(* CODESYS project ST_MUX.project

Project tree, tasks and I/O mapping:
  Device : AC702, Shenzhen Inovance Technology Co., Ltd., version 3.5.11.51
    application Application
      libraries: Standard, * (System)
      task MainTask (cyclic, interval 4 ms, priority 2) calls PLC_PRG
      program PLC_PRG [ST]
      DifferentialMonitor
    HardWare Configuration
    Network Configuration
    Device Diagnosis
    Resources List
    ConfigStorage
    SoftMotion General Axis Pool
    LocalHSIO : 本地高速IO, 汇川技术股份有限公司, version 1.0.0.0
        unmapped channels: DigitalInput, DigitalOutput
    MODBUS_TCP : ModbusTCP本地从站, inovance, version 00.00.00.10
    HwConfiguratioinDevice : SystemConfig, Inovance, version 00.00.00.10
        settings: NetworkConfigArray.NetworkConfigArray.BusType = 10; NetworkConfigArray.NetworkConfigArray.RackSum = 1; NetworkConfigArray.NetworkConfigArray.HardwareConfigArray.HardwareConfigArray.RackNo = 1
*)

// Device/Application/PLC_PRG
PROGRAM PLC_PRG
VAR
	A1: BOOL;
	MUX_R4: REAL;
	A0: BOOL;
	IN2: REAL;
	IN3: REAL;
	IN0: REAL;
	IN1: REAL;
END_VAR

IF A1 THEN
	MUX_R4 := SEL(A0, IN2, IN3);
ELSE
	MUX_R4 := SEL(A0, IN0, IN1);
END_IF;

END_PROGRAM
